{attribute 'no_explicit_call' := 'do not call this function block directly'} 
{attribute 'enable_dynamic_creation'}
FUNCTION_BLOCK PointerListEnumerator EXTENDS Enumerator
VAR
	_ClassName : STRING := __POUNAME();
	_List : IReadOnlyPointerList;
	_Current : PVOID;
END_VAR

{attribute 'monitoring' := 'call'}
PROPERTY ClassName : STRING
GET
ClassName := _ClassName;
END_GET
END_PROPERTY

PROPERTY Current : PVOID
GET
Current := _Current;
END_GET
END_PROPERTY

METHOD INTERNAL Initialize
VAR_INPUT
	list : IReadOnlyPointerList;
END_VAR
_List := list;
END_METHOD

{attribute "object_name" := "MoveNext"}
METHOD MoveNext : BOOL
_CurrentIndex := _CurrentIndex + 1;

IF _CurrentIndex >= _List.Count THEN
	_Current := 0;	
	_CurrentIndex := _List.Count;
ELSE
	_Current := _List.Get(_CurrentIndex);	
	MoveNext := TRUE;
END_IF
END_METHOD

{attribute "object_name" := "Reset"}
METHOD Reset
SUPER^.Reset();

_Current := 0;
END_METHOD

END_FUNCTION_BLOCK

(* stored: Version 1.1.0.1
   POU PointerListEnumerator: Id {6b600d98-a4d1-0f13-3cbb-397b335d25ee}, SpecialFunc None
   Property ClassName: Id {e9cd6f44-c0f7-0035-28b2-789e0b9529af}
   Get Get: Id {c18e11ea-564b-09d7-1c34-99c431ea6204}
   Property Current: Id {96045d59-e34b-0102-15e1-9ba2b60ebccc}
   Get Get: Id {98feb4b4-de08-087c-186e-32093c4e14f3}
   Method Initialize: Id {2b7baa46-574a-041a-287e-45a2e3e8227d}
   Method MoveNext: Id {ad22e0f3-eb62-01b3-3a7f-d684c73f59e9}
   Method Reset: Id {298846f1-921c-0987-0d7b-d675d72bc0b4} *)
